Staubli VAL3: clkValvePage.pgx

program clkValvePage()
begin
  userPage("valves")
end
